PROGRAM Main
VAR
    KlaarVoorBier : BOOL;
    KlaarVoorSpel : BOOL;
END_VAR


KlaarVoorBier := Aangekomen;
KlaarVoorSpel := (Biertjes >= 3);

END_PROGRAM

(* stored: Version 1.1.0.1, ProductVersion 3.1.4024.15
   POU Main: Id {2eff0738-9ba1-4265-99a1-eaec03d7774a}, SpecialFunc None *)
